GLOBALCONSTANTS DefaultPool_AIC_2P_Numeric (* Numeric object pool constants (ID, Scale, Offset, Decimals) *)
  PACKAGE Uebungen::const::UT::AIC;
  VAR_GLOBAL CONSTANT
    InputNumber_AIC_I01_ZERO_N : logiBUS::utils::conversion::phys::NumericObjectPool_S := (u16ObjId := 9000, r32Scale := 0.1, i32Offset := -1000, u8Decimals := 1);
    InputNumber_AIC_I01_SPAN_N : logiBUS::utils::conversion::phys::NumericObjectPool_S := (u16ObjId := 9001, r32Scale := 0.1, i32Offset := -1000, u8Decimals := 1);
    InputNumber_AIC_I02_ZERO_N : logiBUS::utils::conversion::phys::NumericObjectPool_S := (u16ObjId := 9002, r32Scale := 0.1, i32Offset := -1000, u8Decimals := 1);
    InputNumber_AIC_I02_SPAN_N : logiBUS::utils::conversion::phys::NumericObjectPool_S := (u16ObjId := 9003, r32Scale := 0.1, i32Offset := -1000, u8Decimals := 1);
    InputNumber_AIC_I03_ZERO_N : logiBUS::utils::conversion::phys::NumericObjectPool_S := (u16ObjId := 9004, r32Scale := 0.1, i32Offset := -1000, u8Decimals := 1);
    InputNumber_AIC_I03_SPAN_N : logiBUS::utils::conversion::phys::NumericObjectPool_S := (u16ObjId := 9005, r32Scale := 0.1, i32Offset := -1000, u8Decimals := 1);
    InputNumber_AIC_I04_ZERO_N : logiBUS::utils::conversion::phys::NumericObjectPool_S := (u16ObjId := 9006, r32Scale := 0.1, i32Offset := -1000, u8Decimals := 1);
    InputNumber_AIC_I04_SPAN_N : logiBUS::utils::conversion::phys::NumericObjectPool_S := (u16ObjId := 9007, r32Scale := 0.1, i32Offset := -1000, u8Decimals := 1);
    InputNumber_AIC_I05_ZERO_N : logiBUS::utils::conversion::phys::NumericObjectPool_S := (u16ObjId := 9008, r32Scale := 0.1, i32Offset := -1000, u8Decimals := 1);
    InputNumber_AIC_I05_SPAN_N : logiBUS::utils::conversion::phys::NumericObjectPool_S := (u16ObjId := 9009, r32Scale := 0.1, i32Offset := -1000, u8Decimals := 1);
    InputNumber_AIC_I06_ZERO_N : logiBUS::utils::conversion::phys::NumericObjectPool_S := (u16ObjId := 9010, r32Scale := 0.1, i32Offset := -1000, u8Decimals := 1);
    InputNumber_AIC_I06_SPAN_N : logiBUS::utils::conversion::phys::NumericObjectPool_S := (u16ObjId := 9011, r32Scale := 0.1, i32Offset := -1000, u8Decimals := 1);
    InputNumber_AIC_I07_ZERO_N : logiBUS::utils::conversion::phys::NumericObjectPool_S := (u16ObjId := 9012, r32Scale := 0.1, i32Offset := -1000, u8Decimals := 1);
    InputNumber_AIC_I07_SPAN_N : logiBUS::utils::conversion::phys::NumericObjectPool_S := (u16ObjId := 9013, r32Scale := 0.1, i32Offset := -1000, u8Decimals := 1);
    InputNumber_AIC_I08_ZERO_N : logiBUS::utils::conversion::phys::NumericObjectPool_S := (u16ObjId := 9014, r32Scale := 0.1, i32Offset := -1000, u8Decimals := 1);
    InputNumber_AIC_I08_SPAN_N : logiBUS::utils::conversion::phys::NumericObjectPool_S := (u16ObjId := 9015, r32Scale := 0.1, i32Offset := -1000, u8Decimals := 1);
    OutputNumber_c1_N : logiBUS::utils::conversion::phys::NumericObjectPool_S := (u16ObjId := 12001, r32Scale := 1.0, i32Offset := 0, u8Decimals := 0);
    OutputNumber_c9_N : logiBUS::utils::conversion::phys::NumericObjectPool_S := (u16ObjId := 12009, r32Scale := 1.0, i32Offset := 0, u8Decimals := 0);
    OutputNumber_c10_N : logiBUS::utils::conversion::phys::NumericObjectPool_S := (u16ObjId := 12010, r32Scale := 1.0, i32Offset := 0, u8Decimals := 0);
    OutputNumber_c11_N : logiBUS::utils::conversion::phys::NumericObjectPool_S := (u16ObjId := 12011, r32Scale := 1.0, i32Offset := 0, u8Decimals := 0);
    OutputNumber_c12_N : logiBUS::utils::conversion::phys::NumericObjectPool_S := (u16ObjId := 12012, r32Scale := 1.0, i32Offset := 0, u8Decimals := 0);
    OutputNumber_c2_N : logiBUS::utils::conversion::phys::NumericObjectPool_S := (u16ObjId := 12013, r32Scale := 1.0, i32Offset := 0, u8Decimals := 0);
    OutputNumber_c3_N : logiBUS::utils::conversion::phys::NumericObjectPool_S := (u16ObjId := 12014, r32Scale := 1.0, i32Offset := 0, u8Decimals := 0);
    OutputNumber_c4_N : logiBUS::utils::conversion::phys::NumericObjectPool_S := (u16ObjId := 12015, r32Scale := 1.0, i32Offset := 0, u8Decimals := 0);
    OutputNumber_c5_N : logiBUS::utils::conversion::phys::NumericObjectPool_S := (u16ObjId := 12016, r32Scale := 1.0, i32Offset := 0, u8Decimals := 0);
    OutputNumber_c6_N : logiBUS::utils::conversion::phys::NumericObjectPool_S := (u16ObjId := 12017, r32Scale := 1.0, i32Offset := 0, u8Decimals := 0);
    OutputNumber_c7_N : logiBUS::utils::conversion::phys::NumericObjectPool_S := (u16ObjId := 12018, r32Scale := 1.0, i32Offset := 0, u8Decimals := 0);
    OutputNumber_c8_N : logiBUS::utils::conversion::phys::NumericObjectPool_S := (u16ObjId := 12019, r32Scale := 1.0, i32Offset := 0, u8Decimals := 0);
    OutputNumber_Tick_N : logiBUS::utils::conversion::phys::NumericObjectPool_S := (u16ObjId := 12020, r32Scale := 1.0, i32Offset := 0, u8Decimals := 0);
    OutputNumber_AIC_I01_RAW_N : logiBUS::utils::conversion::phys::NumericObjectPool_S := (u16ObjId := 12021, r32Scale := 1.0, i32Offset := 0, u8Decimals := 0);
    OutputNumber_AIC_I01_CAL_N : logiBUS::utils::conversion::phys::NumericObjectPool_S := (u16ObjId := 12022, r32Scale := 1.0, i32Offset := 0, u8Decimals := 1);
    OutputNumber_AIC_I02_RAW_N : logiBUS::utils::conversion::phys::NumericObjectPool_S := (u16ObjId := 12023, r32Scale := 1.0, i32Offset := 0, u8Decimals := 0);
    OutputNumber_AIC_I02_CAL_N : logiBUS::utils::conversion::phys::NumericObjectPool_S := (u16ObjId := 12024, r32Scale := 1.0, i32Offset := 0, u8Decimals := 1);
    OutputNumber_AIC_I03_RAW_N : logiBUS::utils::conversion::phys::NumericObjectPool_S := (u16ObjId := 12025, r32Scale := 1.0, i32Offset := 0, u8Decimals := 0);
    OutputNumber_AIC_I03_CAL_N : logiBUS::utils::conversion::phys::NumericObjectPool_S := (u16ObjId := 12026, r32Scale := 1.0, i32Offset := 0, u8Decimals := 1);
    OutputNumber_AIC_I04_RAW_N : logiBUS::utils::conversion::phys::NumericObjectPool_S := (u16ObjId := 12027, r32Scale := 1.0, i32Offset := 0, u8Decimals := 0);
    OutputNumber_AIC_I04_CAL_N : logiBUS::utils::conversion::phys::NumericObjectPool_S := (u16ObjId := 12028, r32Scale := 1.0, i32Offset := 0, u8Decimals := 1);
    OutputNumber_AIC_I05_RAW_N : logiBUS::utils::conversion::phys::NumericObjectPool_S := (u16ObjId := 12029, r32Scale := 1.0, i32Offset := 0, u8Decimals := 0);
    OutputNumber_AIC_I05_CAL_N : logiBUS::utils::conversion::phys::NumericObjectPool_S := (u16ObjId := 12030, r32Scale := 1.0, i32Offset := 0, u8Decimals := 1);
    OutputNumber_AIC_I06_RAW_N : logiBUS::utils::conversion::phys::NumericObjectPool_S := (u16ObjId := 12031, r32Scale := 1.0, i32Offset := 0, u8Decimals := 0);
    OutputNumber_AIC_I06_CAL_N : logiBUS::utils::conversion::phys::NumericObjectPool_S := (u16ObjId := 12032, r32Scale := 1.0, i32Offset := 0, u8Decimals := 1);
    OutputNumber_AIC_I07_RAW_N : logiBUS::utils::conversion::phys::NumericObjectPool_S := (u16ObjId := 12033, r32Scale := 1.0, i32Offset := 0, u8Decimals := 0);
    OutputNumber_AIC_I07_CAL_N : logiBUS::utils::conversion::phys::NumericObjectPool_S := (u16ObjId := 12034, r32Scale := 1.0, i32Offset := 0, u8Decimals := 1);
    OutputNumber_AIC_I08_RAW_N : logiBUS::utils::conversion::phys::NumericObjectPool_S := (u16ObjId := 12035, r32Scale := 1.0, i32Offset := 0, u8Decimals := 0);
    OutputNumber_AIC_I08_CAL_N : logiBUS::utils::conversion::phys::NumericObjectPool_S := (u16ObjId := 12036, r32Scale := 1.0, i32Offset := 0, u8Decimals := 1);
    OutputNumber_AIC_I01_ZERORAW_N : logiBUS::utils::conversion::phys::NumericObjectPool_S := (u16ObjId := 12037, r32Scale := 1.0, i32Offset := 0, u8Decimals := 0);
    OutputNumber_AIC_I01_SPANRAW_N : logiBUS::utils::conversion::phys::NumericObjectPool_S := (u16ObjId := 12038, r32Scale := 1.0, i32Offset := 0, u8Decimals := 0);
    OutputNumber_AIC_I02_ZERORAW_N : logiBUS::utils::conversion::phys::NumericObjectPool_S := (u16ObjId := 12039, r32Scale := 1.0, i32Offset := 0, u8Decimals := 0);
    OutputNumber_AIC_I02_SPANRAW_N : logiBUS::utils::conversion::phys::NumericObjectPool_S := (u16ObjId := 12040, r32Scale := 1.0, i32Offset := 0, u8Decimals := 0);
    OutputNumber_AIC_I03_ZERORAW_N : logiBUS::utils::conversion::phys::NumericObjectPool_S := (u16ObjId := 12041, r32Scale := 1.0, i32Offset := 0, u8Decimals := 0);
    OutputNumber_AIC_I03_SPANRAW_N : logiBUS::utils::conversion::phys::NumericObjectPool_S := (u16ObjId := 12042, r32Scale := 1.0, i32Offset := 0, u8Decimals := 0);
    OutputNumber_AIC_I04_ZERORAW_N : logiBUS::utils::conversion::phys::NumericObjectPool_S := (u16ObjId := 12043, r32Scale := 1.0, i32Offset := 0, u8Decimals := 0);
    OutputNumber_AIC_I04_SPANRAW_N : logiBUS::utils::conversion::phys::NumericObjectPool_S := (u16ObjId := 12044, r32Scale := 1.0, i32Offset := 0, u8Decimals := 0);
    OutputNumber_AIC_I05_ZERORAW_N : logiBUS::utils::conversion::phys::NumericObjectPool_S := (u16ObjId := 12045, r32Scale := 1.0, i32Offset := 0, u8Decimals := 0);
    OutputNumber_AIC_I05_SPANRAW_N : logiBUS::utils::conversion::phys::NumericObjectPool_S := (u16ObjId := 12046, r32Scale := 1.0, i32Offset := 0, u8Decimals := 0);
    OutputNumber_AIC_I06_ZERORAW_N : logiBUS::utils::conversion::phys::NumericObjectPool_S := (u16ObjId := 12047, r32Scale := 1.0, i32Offset := 0, u8Decimals := 0);
    OutputNumber_AIC_I06_SPANRAW_N : logiBUS::utils::conversion::phys::NumericObjectPool_S := (u16ObjId := 12048, r32Scale := 1.0, i32Offset := 0, u8Decimals := 0);
    OutputNumber_AIC_I07_ZERORAW_N : logiBUS::utils::conversion::phys::NumericObjectPool_S := (u16ObjId := 12049, r32Scale := 1.0, i32Offset := 0, u8Decimals := 0);
    OutputNumber_AIC_I07_SPANRAW_N : logiBUS::utils::conversion::phys::NumericObjectPool_S := (u16ObjId := 12050, r32Scale := 1.0, i32Offset := 0, u8Decimals := 0);
    OutputNumber_AIC_I08_ZERORAW_N : logiBUS::utils::conversion::phys::NumericObjectPool_S := (u16ObjId := 12051, r32Scale := 1.0, i32Offset := 0, u8Decimals := 0);
    OutputNumber_AIC_I08_SPANRAW_N : logiBUS::utils::conversion::phys::NumericObjectPool_S := (u16ObjId := 12052, r32Scale := 1.0, i32Offset := 0, u8Decimals := 0);
    NumberVariable_AIC_RAW_I01_N : logiBUS::utils::conversion::phys::NumericObjectPool_S := (u16ObjId := 21000, r32Scale := 1.0, i32Offset := 0, u8Decimals := 0);
    NumberVariable_AIC_RAW_I02_N : logiBUS::utils::conversion::phys::NumericObjectPool_S := (u16ObjId := 21001, r32Scale := 1.0, i32Offset := 0, u8Decimals := 0);
    NumberVariable_AIC_RAW_I03_N : logiBUS::utils::conversion::phys::NumericObjectPool_S := (u16ObjId := 21002, r32Scale := 1.0, i32Offset := 0, u8Decimals := 0);
    NumberVariable_AIC_RAW_I04_N : logiBUS::utils::conversion::phys::NumericObjectPool_S := (u16ObjId := 21003, r32Scale := 1.0, i32Offset := 0, u8Decimals := 0);
    NumberVariable_AIC_RAW_I05_N : logiBUS::utils::conversion::phys::NumericObjectPool_S := (u16ObjId := 21004, r32Scale := 1.0, i32Offset := 0, u8Decimals := 0);
    NumberVariable_AIC_RAW_I06_N : logiBUS::utils::conversion::phys::NumericObjectPool_S := (u16ObjId := 21005, r32Scale := 1.0, i32Offset := 0, u8Decimals := 0);
    NumberVariable_AIC_RAW_I07_N : logiBUS::utils::conversion::phys::NumericObjectPool_S := (u16ObjId := 21006, r32Scale := 1.0, i32Offset := 0, u8Decimals := 0);
    NumberVariable_AIC_RAW_I08_N : logiBUS::utils::conversion::phys::NumericObjectPool_S := (u16ObjId := 21007, r32Scale := 1.0, i32Offset := 0, u8Decimals := 0);
    NumberVariable_AIC_CAL_I01_N : logiBUS::utils::conversion::phys::NumericObjectPool_S := (u16ObjId := 21008, r32Scale := 1.0, i32Offset := 0, u8Decimals := 1);
    NumberVariable_AIC_CAL_I02_N : logiBUS::utils::conversion::phys::NumericObjectPool_S := (u16ObjId := 21009, r32Scale := 1.0, i32Offset := 0, u8Decimals := 1);
    NumberVariable_AIC_CAL_I03_N : logiBUS::utils::conversion::phys::NumericObjectPool_S := (u16ObjId := 21010, r32Scale := 1.0, i32Offset := 0, u8Decimals := 1);
    NumberVariable_AIC_CAL_I04_N : logiBUS::utils::conversion::phys::NumericObjectPool_S := (u16ObjId := 21011, r32Scale := 1.0, i32Offset := 0, u8Decimals := 1);
    NumberVariable_AIC_CAL_I05_N : logiBUS::utils::conversion::phys::NumericObjectPool_S := (u16ObjId := 21012, r32Scale := 1.0, i32Offset := 0, u8Decimals := 1);
    NumberVariable_AIC_CAL_I06_N : logiBUS::utils::conversion::phys::NumericObjectPool_S := (u16ObjId := 21013, r32Scale := 1.0, i32Offset := 0, u8Decimals := 1);
    NumberVariable_AIC_CAL_I07_N : logiBUS::utils::conversion::phys::NumericObjectPool_S := (u16ObjId := 21014, r32Scale := 1.0, i32Offset := 0, u8Decimals := 1);
    NumberVariable_AIC_CAL_I08_N : logiBUS::utils::conversion::phys::NumericObjectPool_S := (u16ObjId := 21015, r32Scale := 1.0, i32Offset := 0, u8Decimals := 1);
    NumberVariable_AIC_I01_ZERO_N : logiBUS::utils::conversion::phys::NumericObjectPool_S := (u16ObjId := 21016, r32Scale := 0.1, i32Offset := -1000, u8Decimals := 1);
    NumberVariable_AIC_I01_SPAN_N : logiBUS::utils::conversion::phys::NumericObjectPool_S := (u16ObjId := 21017, r32Scale := 0.1, i32Offset := -1000, u8Decimals := 1);
    NumberVariable_AIC_I02_ZERO_N : logiBUS::utils::conversion::phys::NumericObjectPool_S := (u16ObjId := 21018, r32Scale := 0.1, i32Offset := -1000, u8Decimals := 1);
    NumberVariable_AIC_I02_SPAN_N : logiBUS::utils::conversion::phys::NumericObjectPool_S := (u16ObjId := 21019, r32Scale := 0.1, i32Offset := -1000, u8Decimals := 1);
    NumberVariable_AIC_I03_ZERO_N : logiBUS::utils::conversion::phys::NumericObjectPool_S := (u16ObjId := 21020, r32Scale := 0.1, i32Offset := -1000, u8Decimals := 1);
    NumberVariable_AIC_I03_SPAN_N : logiBUS::utils::conversion::phys::NumericObjectPool_S := (u16ObjId := 21021, r32Scale := 0.1, i32Offset := -1000, u8Decimals := 1);
    NumberVariable_AIC_I04_ZERO_N : logiBUS::utils::conversion::phys::NumericObjectPool_S := (u16ObjId := 21022, r32Scale := 0.1, i32Offset := -1000, u8Decimals := 1);
    NumberVariable_AIC_I04_SPAN_N : logiBUS::utils::conversion::phys::NumericObjectPool_S := (u16ObjId := 21023, r32Scale := 0.1, i32Offset := -1000, u8Decimals := 1);
    NumberVariable_AIC_I05_ZERO_N : logiBUS::utils::conversion::phys::NumericObjectPool_S := (u16ObjId := 21024, r32Scale := 0.1, i32Offset := -1000, u8Decimals := 1);
    NumberVariable_AIC_I05_SPAN_N : logiBUS::utils::conversion::phys::NumericObjectPool_S := (u16ObjId := 21025, r32Scale := 0.1, i32Offset := -1000, u8Decimals := 1);
    NumberVariable_AIC_I06_ZERO_N : logiBUS::utils::conversion::phys::NumericObjectPool_S := (u16ObjId := 21026, r32Scale := 0.1, i32Offset := -1000, u8Decimals := 1);
    NumberVariable_AIC_I06_SPAN_N : logiBUS::utils::conversion::phys::NumericObjectPool_S := (u16ObjId := 21027, r32Scale := 0.1, i32Offset := -1000, u8Decimals := 1);
    NumberVariable_AIC_I07_ZERO_N : logiBUS::utils::conversion::phys::NumericObjectPool_S := (u16ObjId := 21028, r32Scale := 0.1, i32Offset := -1000, u8Decimals := 1);
    NumberVariable_AIC_I07_SPAN_N : logiBUS::utils::conversion::phys::NumericObjectPool_S := (u16ObjId := 21029, r32Scale := 0.1, i32Offset := -1000, u8Decimals := 1);
    NumberVariable_AIC_I08_ZERO_N : logiBUS::utils::conversion::phys::NumericObjectPool_S := (u16ObjId := 21030, r32Scale := 0.1, i32Offset := -1000, u8Decimals := 1);
    NumberVariable_AIC_I08_SPAN_N : logiBUS::utils::conversion::phys::NumericObjectPool_S := (u16ObjId := 21031, r32Scale := 0.1, i32Offset := -1000, u8Decimals := 1);
    NumberVariable_AIC_I01_ZERORAW_N : logiBUS::utils::conversion::phys::NumericObjectPool_S := (u16ObjId := 21032, r32Scale := 1.0, i32Offset := 0, u8Decimals := 0);
    NumberVariable_AIC_I01_SPANRAW_N : logiBUS::utils::conversion::phys::NumericObjectPool_S := (u16ObjId := 21033, r32Scale := 1.0, i32Offset := 0, u8Decimals := 0);
    NumberVariable_AIC_I02_ZERORAW_N : logiBUS::utils::conversion::phys::NumericObjectPool_S := (u16ObjId := 21034, r32Scale := 1.0, i32Offset := 0, u8Decimals := 0);
    NumberVariable_AIC_I02_SPANRAW_N : logiBUS::utils::conversion::phys::NumericObjectPool_S := (u16ObjId := 21035, r32Scale := 1.0, i32Offset := 0, u8Decimals := 0);
    NumberVariable_AIC_I03_ZERORAW_N : logiBUS::utils::conversion::phys::NumericObjectPool_S := (u16ObjId := 21036, r32Scale := 1.0, i32Offset := 0, u8Decimals := 0);
    NumberVariable_AIC_I03_SPANRAW_N : logiBUS::utils::conversion::phys::NumericObjectPool_S := (u16ObjId := 21037, r32Scale := 1.0, i32Offset := 0, u8Decimals := 0);
    NumberVariable_AIC_I04_ZERORAW_N : logiBUS::utils::conversion::phys::NumericObjectPool_S := (u16ObjId := 21038, r32Scale := 1.0, i32Offset := 0, u8Decimals := 0);
    NumberVariable_AIC_I04_SPANRAW_N : logiBUS::utils::conversion::phys::NumericObjectPool_S := (u16ObjId := 21039, r32Scale := 1.0, i32Offset := 0, u8Decimals := 0);
    NumberVariable_AIC_I05_ZERORAW_N : logiBUS::utils::conversion::phys::NumericObjectPool_S := (u16ObjId := 21040, r32Scale := 1.0, i32Offset := 0, u8Decimals := 0);
    NumberVariable_AIC_I05_SPANRAW_N : logiBUS::utils::conversion::phys::NumericObjectPool_S := (u16ObjId := 21041, r32Scale := 1.0, i32Offset := 0, u8Decimals := 0);
    NumberVariable_AIC_I06_ZERORAW_N : logiBUS::utils::conversion::phys::NumericObjectPool_S := (u16ObjId := 21042, r32Scale := 1.0, i32Offset := 0, u8Decimals := 0);
    NumberVariable_AIC_I06_SPANRAW_N : logiBUS::utils::conversion::phys::NumericObjectPool_S := (u16ObjId := 21043, r32Scale := 1.0, i32Offset := 0, u8Decimals := 0);
    NumberVariable_AIC_I07_ZERORAW_N : logiBUS::utils::conversion::phys::NumericObjectPool_S := (u16ObjId := 21044, r32Scale := 1.0, i32Offset := 0, u8Decimals := 0);
    NumberVariable_AIC_I07_SPANRAW_N : logiBUS::utils::conversion::phys::NumericObjectPool_S := (u16ObjId := 21045, r32Scale := 1.0, i32Offset := 0, u8Decimals := 0);
    NumberVariable_AIC_I08_ZERORAW_N : logiBUS::utils::conversion::phys::NumericObjectPool_S := (u16ObjId := 21046, r32Scale := 1.0, i32Offset := 0, u8Decimals := 0);
    NumberVariable_AIC_I08_SPANRAW_N : logiBUS::utils::conversion::phys::NumericObjectPool_S := (u16ObjId := 21047, r32Scale := 1.0, i32Offset := 0, u8Decimals := 0);
  END_VAR
END_GLOBALCONSTANTS
